PROGRAM MainParComfer_HMI
VAR
END_VAR

MainFramDUT.ComName:='GIDEON';//公司名称;
MainFramDUT.ProjectName:='ICP_01';//项目名称	
MainFramDUT.ShowTime:=g_SystemTime;//当前时间显示变量
//按钮灯
MainFramDUT.StartLamp:=fbMachineState.StartLamp;//启面急停动指示
MainFramDUT.ResetLamp:=fbMachineState.ResetLamp;//复面急停位指示
MainFramDUT.StopLamp:=fbMachineState.StopLamp;//停面急停止，报错指示
	
fbMachineState.HMI_E_Stop:=MainFramDUT.E_Stop;//界面急停显示
fbMachineState.HMI_Start:=MainFramDUT.Start;//界面启动
fbMachineState.HMI_Reset:=MainFramDUT.Reset;//界面复位
fbMachineState.HMI_Stop:=MainFramDUT.Stop;//界面停止
//三色灯
MainFramDUT.GreenLamp:=fbMachineState.GreenLamp;//绿灯
MainFramDUT.RedLamp:=fbMachineState.RedLamp;//红灯
MainFramDUT.YellowLamp:=fbMachineState.YellowLamp;//黄灯
//MainFramDUT.Loading:=;//界面登录
//MainFramDUT.Quit:=;//界面退出
MainFramDUT.versions:=gVersion;//版本号传递
MainFramDUT.RunStateTxt:=fbMachineState.RunStateTxtS;//版本号传递
MainFramDUT.ErrWTxtShow:=gErrWTxtShow;//版本号传递

END_PROGRAM

(* stored: Version 1.1.0.1, ProductVersion 3.1.4024.4
   POU MainParComfer_HMI: Id {f84b23e7-df2a-469e-aea3-f3048715a0cb}, SpecialFunc None *)
